// TIA Portal V21 export
VAR_GLOBAL   // PLC tag table "KAllZona"
END_VAR
VAR_GLOBAL CONSTANT   // user constants
   KAllZona_CentralinaSicurezza : Int := 1;
   KAllZona_PressostatoGenerale : Int := 3;
   KAllZona_CicloNonInserito : Int := 2;
END_VAR
